{attribute 'qualified_only'}
VAR_GLOBAL
	bGreenLED AT %Q* : BOOL;
	bRedLED AT %Q* : BOOL;
	
	stWinchValveOutput : ST_ValveOutput;
	stCylValveOutput : ST_ValveOutput;
END_VAR

(* stored: Version 1.1.0.1, ProductVersion 3.1.4024.12
   GVL G_Outputs: Id {678ea39b-1e41-4c00-a687-e80f05b2794d} *)
